(* IEC 61131-3 sources: Project_Icarus/d4ryus, 2 files *)

(* ---- test.st ---- *)
PRORAMM blub
VAR
	var1:INT := 3;
	var2:BOOL := TRUE;
	var3:REAL;
END_VAR

PRINT(var1---var2---var3);

(* bvlubljasldjf *)

IF (3 > 5)       (********************)
THEN             (* a then statement *)
    PRINT(blub); (* the then block   *)
END_IF           (********************)

IF (var2)
THEN
	PRINT(great_job_sir);
END_IF

END_PROGRAM

 (* aslkjf *)

(* ---- test_preprozessed.st ---- *)
IF(3+4>5)§THEN§blub§END_IF§END_PROGRAM
01234567890123456789012345678901234567890
